ABB RAPID module: TCP_mtip_on_mmtool.mod

MODULE TCP_mtip_on_mmtool
	! Points are read in order of declaration.
  ! Please do not change the order of points!

  LOCAL PERS robtarget pTCP_Point1:=[[1039.458,-180.2702,1049.362],[0.00115850940346718,0.25465190410614,-0.967029690742493,0.00216152798384428],[-1,-1,-1,0],[9E+09,9E+09,9E+09,9E+09,9E+09,9E+09]];
	LOCAL PERS robtarget pTCP_Point2:=[[1171.878,-415.3574,984.5333],[0.0586728490889072,0.247810930013657,-0.942488789558411,-0.216476634144783],[-1,0,-1,0],[9E+09,9E+09,9E+09,9E+09,9E+09,9E+09]];
	LOCAL PERS robtarget pTCP_Point3:=[[911.2497,-528.2729,922.6545],[0.165729492902756,-0.189653649926186,0.929665446281433,0.268863141536713],[-1,0,-1,0],[9E+09,9E+09,9E+09,9E+09,9E+09,9E+09]];
	LOCAL PERS robtarget pTCP_Point4:=[[901.7825,89.03639,973.4263],[0.0705400928854942,-0.175300568342209,0.95093309879303,-0.244989961385727],[0,-1,0,0],[9E+09,9E+09,9E+09,9E+09,9E+09,9E+09]];
	LOCAL PERS robtarget pTCP_Point5:=[[1285.833,96.4272,927.3226],[0.242517322301865,0.12230172008276,-0.939350545406342,0.209399700164795],[0,-1,-1,0],[9E+09,9E+09,9E+09,9E+09,9E+09,9E+09]];
	LOCAL PERS robtarget pTCP_Point6:=[[1347.79,-203.7098,964.2482],[0.260562598705292,0.084771029651165,-0.960877299308777,-0.040445052087307],[-1,-1,-1,0],[9E+09,9E+09,9E+09,9E+09,9E+09,9E+09]];
	LOCAL PERS robtarget pTCP_Point7:=[[953.6797,-144.8428,1043.09],[0.0410320535302162,-0.610346674919128,0.788216829299927,-0.0671382024884224],[-1,-1,-1,0],[9E+09,9E+09,9E+09,9E+09,9E+09,9E+09]];

ENDMODULE
